// TIA Portal V18 export
DATA_BLOCK "LGF_FIFO_DB"   // DB285
AUTHOR : Siemens_Industry_Support
FAMILY : LGF
NAME : LGF_FIFO
VERSION : 0.1
// stored: AutoNumber true, DBAccessibleFromOPCUA true, InstanceOfName LGF_FIFO, InstanceOfType FB
"LGF_FIFO"
   // VAR_INPUT
   //    enqueue : Bool;
   //    dequeue : Bool;
   //    reset : Bool;
   //    clear : Bool;
   //    initialItem : Variant;
   // END_VAR
   // VAR_OUTPUT
   //    error { ExternalWritable := 'False'} : Bool;
   //    status { ExternalWritable := 'False'} : Word;
   //    subFunctionStatus { ExternalWritable := 'False'} : Word;
   //    elementCount { ExternalWritable := 'False'} : DInt;
   //    isEmpty { ExternalWritable := 'False'} : Bool;
   // END_VAR
   // VAR_IN_OUT
   //    item : Variant;
   //    buffer : Variant;
   // END_VAR
   // VAR
   //    statEdgesMem { ExternalAccessible := 'False'; ExternalVisible := 'False'; ExternalWritable := 'False'} : Struct
   //       enqueue { ExternalAccessible := 'False'; ExternalVisible := 'False'; ExternalWritable := 'False'} : Bool;
   //       dequeue { ExternalAccessible := 'False'; ExternalVisible := 'False'; ExternalWritable := 'False'} : Bool;
   //       clear { ExternalAccessible := 'False'; ExternalVisible := 'False'; ExternalWritable := 'False'} : Bool;
   //    END_STRUCT;
   //    statFirstItemIndex { ExternalAccessible := 'False'; ExternalVisible := 'False'; ExternalWritable := 'False'} : Int;
   //    statNextEmptyItemIndex { ExternalAccessible := 'False'; ExternalVisible := 'False'; ExternalWritable := 'False'} : Int;
   //    statElementCount { ExternalAccessible := 'False'; ExternalVisible := 'False'; ExternalWritable := 'False'} : DInt;
   // END_VAR
BEGIN
END_DATA_BLOCK
